// TwinCAT 3 PLC project TcTcpUdpRT_Test
// ProgramVersion: 3.1.4026.20
// libraries:
//   Tc2_Standard, * (Beckhoff Automation GmbH)
//   Tc2_System, * (Beckhoff Automation GmbH)
//   [TcTcpUdpRT], * (TcInterfaces)
//   TcUnit, * (www.tcunit.org)
// project tree:
//   / PlcTask.TcTTO, PRG_TEST.TcPOU (not stored)
//   TESTs/ ArpPing_Test.TcPOU (not stored), RingBuffer_Test.TcPOU, TcpClient_Test.TcPOU, TcpServer_Test.TcPOU, UdpSendReceive_Test.TcPOU
// real-time tasks:
//   TASK PlcTask: cycle T#1ms, priority 6, ADS port 350
// I/O:
//   DEVICE EthernetRT (RT-Ethernet Adapter)

CONFIGURATION TcTcpUdpRT_Test
    RESOURCE PLC ON TwinCAT3
        TASK PlcTask(INTERVAL := T#1ms, PRIORITY := 6);
        PROGRAM PRG_TEST WITH PlcTask : PRG_TEST;
    END_RESOURCE
END_CONFIGURATION

// ---- TESTs/RingBuffer_Test.TcPOU
FUNCTION_BLOCK RingBuffer_Test EXTENDS FB_TestSuite
VAR
	RingBuf: RingBuffer;
	RingBufUnallocated: RingBuffer;  // Init() is never called on this instance, used for the unallocated corner cases
	ReadBuffer: ARRAY[0..(TcTcpUdpRT_Param.RingBufferSize-1)] OF BYTE;
	WriteBuffer: ARRAY[0..(WriteBufferSize-1)] OF BYTE;
	emptyPointer: POINTER TO BYTE;
	bytePointer: BYTE;
END_VAR
VAR CONSTANT
	WriteBufferSize: UDINT := 35000;
END_VAR

IF NOT RingBuf.IsAllocated THEN
	RingBuf.Init(BufferSize:= TcTcpUdpRT_Param.RingBufferSize);  // Allocate once before the tests run
END_IF

//WriteWithNoDataPointer();
//WriteWithNoDataLength();
//ReadWithNoDataPointer();
//ReadWithNoDataLength();

Write3kToBufferAndEmptyIt();
ExpectBufferToBeEmpty();
ReadFromEmptyBuffer();
Write1kBytesToBuffer();
ExpectBufferNotToEmpty();

Read2kBytesFrom1kBytesBuffer();
Write25kMoreBytesToBuffer();
ExpectBufferToNotBeFull();

Read24kMoreBytesFromBuffer();
Write8kMoreBytesToBufferAndWrapAround();
Read10kMoreBytesAndWrapAround();

WriteOverflowBuffer();
WriteFullSizeOfBuffer();
ExpectBufferToBeFull();
Write1ByteOverWrapAroundAndRead1ByteOver();

// Corner cases on a buffer that was never allocated
UnallocatedBufferState();
ReadFromUnallocatedBuffer();
WriteToUnallocatedBuffer();
EmptyUnallocatedBuffer();
InitUnallocatedBufferWithDefaultSize();

METHOD EmptyUnallocatedBuffer
VAR
	Emptied: BOOL;
END_VAR
IF TEST_ORDERED('EmptyUnallocatedBuffer') THEN
	Emptied := RingBufUnallocated.EmptyBuffer();
	AssertFalse(Condition:= Emptied, Message:= 'Expected EmptyBuffer to return FALSE on an unallocated buffer');
	AssertTrue(Condition:= RingBufUnallocated.Error, Message:= 'Expected an error when emptying an unallocated buffer');
	AssertEquals_STRING(Expected:= 'Ring buffer is not allocated, call Init() first', Actual:= RingBufUnallocated.GetError, Message:= 'Unexpected error string when emptying an unallocated buffer');

	RingBufUnallocated.ResetError();
	AssertFalse(Condition:= RingBufUnallocated.Error, Message:= 'Ring buffer did not reset error after emptying unallocated buffer');
	TEST_FINISHED();
END_IF
END_METHOD

METHOD ExpectBufferNotToEmpty
IF TEST_ORDERED('ExpectBufferNotToEmpty') THEN
	AssertFalse(Condition:= RingBuf.IsBufferEmpty, Message:= 'Expected IsBufferEmpty returned TRUE when the buffer was not empty');
	TEST_FINISHED();
END_IF
END_METHOD

METHOD ExpectBufferToBeEmpty
IF TEST_ORDERED('ExpectBufferToBeEmpty') THEN
	RingBuf.EmptyBuffer();
	AssertTrue(Condition:= RingBuf.IsBufferEmpty, Message:= 'Expected IsBufferEmpty returned FALSE when the buffer was empty');
	TEST_FINISHED();
END_IF
END_METHOD

METHOD ExpectBufferToBeFull
IF TEST_ORDERED('ExpectBufferToBeFull') THEN
	AssertTRUE(Condition:= RingBuf.IsBufferFull, Message:= 'Expected IsBufferFull returned FALSE when the buffer was full');
	TEST_FINISHED();
END_IF
END_METHOD

METHOD ExpectBufferToNotBeFull
IF TEST_ORDERED('ExpectBufferToNotBeFull') THEN
	AssertFalse(Condition:= RingBuf.IsBufferFull, Message:= 'Expected IsBufferFull returned TRUE when the buffer was not full');
	TEST_FINISHED();
END_IF
END_METHOD

METHOD InitUnallocatedBufferWithDefaultSize
VAR
	DataChar: BYTE := 7;
	DataSize: UDINT := 10;
	Initialized: BOOL;
	Written: UDINT;
	Read: UDINT;
END_VAR
IF TEST_ORDERED('InitUnallocatedBufferWithDefaultSize') THEN
	// Init with size 0 falls back to the default size
	Initialized := RingBufUnallocated.Init(BufferSize:= 0);
	AssertTrue(Condition:= Initialized, Message:= 'Expected Init() with size 0 to allocate the default size');
	AssertFalse(Condition:= RingBufUnallocated.Error, Message:= RingBufUnallocated.GetError);
	AssertTrue(Condition:= RingBufUnallocated.IsAllocated, Message:= 'Expected IsAllocated to be TRUE after Init()');
	AssertEquals_UDINT(Expected:= TcTcpUdpRT_Param.RingBufferSize, Actual:= RingBufUnallocated.Size, Message:= 'Expected Size to be the default size after Init() with size 0');
	AssertTrue(Condition:= RingBufUnallocated.IsBufferEmpty, Message:= 'Expected IsBufferEmpty to be TRUE right after Init()');
	AssertFalse(Condition:= RingBufUnallocated.IsBufferFull, Message:= 'Expected IsBufferFull to be FALSE right after Init()');

	// A second Init must not reallocate or change the size
	Initialized := RingBufUnallocated.Init(BufferSize:= 123);
	AssertTrue(Condition:= Initialized, Message:= 'Expected a second Init() to return TRUE');
	AssertEquals_UDINT(Expected:= TcTcpUdpRT_Param.RingBufferSize, Actual:= RingBufUnallocated.Size, Message:= 'A second Init() changed the size of an already allocated buffer');

	// The buffer is usable after Init()
	MEMSET(destAddr:= ADR(WriteBuffer), fillByte:= DataChar, n:= DataSize);
	MEMSET(destAddr:= ADR(ReadBuffer), fillByte:= 0, n:= TcTcpUdpRT_Param.RingBufferSize);
	Written := RingBufUnallocated.Write(Data:= ADR(WriteBuffer), Length:= DataSize);
	Read := RingBufUnallocated.Read(Data:= ADR(ReadBuffer), Length:= DataSize);
	AssertEquals_UDINT(Expected:= DataSize, Actual:= Written, Message:= 'Written data to the newly allocated buffer does not match');
	AssertEquals_UDINT(Expected:= DataSize, Actual:= Read, Message:= 'Read data from the newly allocated buffer does not match');
	AssertEquals_BYTE(Expected:= DataChar, Actual:= ReadBuffer[DataSize-1], Message:= 'The last element read from the newly allocated buffer was not correct');
	AssertFalse(Condition:= RingBufUnallocated.Error, Message:= RingBufUnallocated.GetError);
	TEST_FINISHED();
END_IF
END_METHOD

METHOD Read10kMoreBytesAndWrapAround
VAR
	DataSize: UDINT := 10000;
	ExpectedSize: UDINT := 9000;
	Read: UDINT;
END_VAR
IF TEST_ORDERED('Read10kMoreBytesAndWrapAround') THEN
	MEMSET(destAddr:= ADR(ReadBuffer), fillByte:= 0, n:= TcTcpUdpRT_Param.RingBufferSize);
	
	Read := RingBuf.Read(Data:= ADR(ReadBuffer), Length:= DataSize);
	AssertEquals_UDINT(Expected:= ExpectedSize, Actual:= Read, Message:= CONCAT('Read data from ring buffer returned a length of ', TO_STRING(Read)));
	AssertTrue(Condition:= ReadBuffer[0] <> 0, Message:= 'The firste element was not different from zero');
	AssertTrue(Condition:= ReadBuffer[ExpectedSize-1] <> 0, Message:= 'The 8999th element was not different from zero');
	AssertTrue(Condition:= ReadBuffer[ExpectedSize] = 0, Message:= 'The 9000th element was not zero');
	AssertTrue(Condition:= ReadBuffer[DataSize] = 0, Message:= 'The last element was not zero');
	TEST_FINISHED();
END_IF
END_METHOD

METHOD Read24kMoreBytesFromBuffer
VAR
	DataSize: UDINT := 24000;
	ExpectedSize: UDINT := 24000;
	Read: UDINT;
END_VAR
IF TEST_ORDERED('Read24kMoreBytesFromBuffer') THEN
	MEMSET(destAddr:= ADR(ReadBuffer), fillByte:= 0, n:= TcTcpUdpRT_Param.RingBufferSize);
	
	Read := RingBuf.Read(Data:= ADR(ReadBuffer), Length:= DataSize);
	AssertEquals_UDINT(Expected:= ExpectedSize, Actual:= Read, Message:= CONCAT('Read data from ring buffer returned a length of ', TO_STRING(Read)));
	AssertTrue(Condition:= ReadBuffer[0] <> 0, Message:= 'The firste element was not different from zero');
	AssertTrue(Condition:= ReadBuffer[18475] <> 0, Message:= 'A random element was not different from zero');
	AssertTrue(Condition:= ReadBuffer[DataSize-1] <> 0, Message:= 'The last element was not different from zero');
	TEST_FINISHED();
END_IF
END_METHOD

METHOD Read2kBytesFrom1kBytesBuffer
VAR
	DataSize: UDINT := 2000;
	ExpectedSize: UDINT := 1000;
	Read: UDINT;
END_VAR
IF TEST_ORDERED('Read2kBytesFrom1kBytesBuffer') THEN
	MEMSET(destAddr:= ADR(ReadBuffer), fillByte:= 0, n:= TcTcpUdpRT_Param.RingBufferSize);
	
	Read := RingBuf.Read(Data:= ADR(ReadBuffer), Length:= DataSize);
	AssertEquals_UDINT(Expected:= ExpectedSize, Actual:= Read, Message:= CONCAT('Read data from ring buffer returned a length of ', TO_STRING(Read)));
	AssertTrue(Condition:= ReadBuffer[0] <> 0, Message:= 'The firste element was not different from zero');
	AssertTrue(Condition:= ReadBuffer[ExpectedSize-1] <> 0, Message:= 'The 999th element was not different from zero');
	AssertTrue(Condition:= ReadBuffer[ExpectedSize] = 0, Message:= 'The 1000th element was not zero');
	AssertTrue(Condition:= ReadBuffer[DataSize-1] = 0, Message:= 'The last element was not zero');
	TEST_FINISHED();
END_IF
END_METHOD

METHOD ReadFromEmptyBuffer
VAR
	DataSize: UDINT := 10;
	ExpectedSize: UDINT := 0;
	Read: UDINT;
END_VAR
IF TEST_ORDERED('ReadFromEmptyBuffer') THEN
	MEMSET(destAddr:= ADR(ReadBuffer), fillByte:= 0, n:= TcTcpUdpRT_Param.RingBufferSize);
	
	Read := RingBuf.Read(Data:= ADR(ReadBuffer), Length:= DataSize);
	AssertEquals_UDINT(Expected:= ExpectedSize, Actual:= Read, Message:= CONCAT('Read data from empty ring buffer returned a length of ', TO_STRING(Read)));
	TEST_FINISHED();
END_IF
END_METHOD

METHOD ReadFromUnallocatedBuffer
VAR
	DataSize: UDINT := 10;
	Read: UDINT;
END_VAR
IF TEST_ORDERED('ReadFromUnallocatedBuffer') THEN
	MEMSET(destAddr:= ADR(ReadBuffer), fillByte:= 0, n:= TcTcpUdpRT_Param.RingBufferSize);

	Read := RingBufUnallocated.Read(Data:= ADR(ReadBuffer), Length:= DataSize);
	AssertEquals_UDINT(Expected:= 0, Actual:= Read, Message:= CONCAT('Read from unallocated ring buffer returned a length of ', TO_STRING(Read)));
	AssertTrue(Condition:= RingBufUnallocated.Error, Message:= 'Expected an error when reading from an unallocated buffer');
	AssertEquals_STRING(Expected:= 'Ring buffer is not allocated, call Init() first', Actual:= RingBufUnallocated.GetError, Message:= 'Unexpected error string when reading from an unallocated buffer');
	AssertEquals_BYTE(Expected:= 0, Actual:= ReadBuffer[0], Message:= 'Read from unallocated buffer modified the destination');

	RingBufUnallocated.ResetError();
	AssertFalse(Condition:= RingBufUnallocated.Error, Message:= 'Ring buffer did not reset error after read from unallocated buffer');
	TEST_FINISHED();
END_IF
END_METHOD

METHOD ReadWithNoDataLength
IF TEST_ORDERED('ReadWithNoDataLength') THEN
	emptyPointer := ADR(bytePointer);
	RingBuf.Read(Data:= emptyPointer, Length:= 0);
	AssertTrue(Condition:= RingBuf.Error, Message:= 'Reading to ring buffer did not handle a data length of zero');
	RingBuf.ResetError();
	TEST_FINISHED();
END_IF
END_METHOD

METHOD ReadWithNoDataPointer
IF TEST_ORDERED('ReadWithNoDataPointer') THEN
	emptyPointer := 0;
	RingBuf.Read(Data:= emptyPointer, Length:= 10);
	AssertTrue(Condition:= RingBuf.Error, Message:= 'Reading to ring buffer did not handle empty data pointer');
	RingBuf.ResetError();
	TEST_FINISHED();
END_IF
END_METHOD

METHOD UnallocatedBufferState
IF TEST_ORDERED('UnallocatedBufferState') THEN
	AssertFalse(Condition:= RingBufUnallocated.IsAllocated, Message:= 'Expected IsAllocated to be FALSE before Init()');
	AssertEquals_UDINT(Expected:= 0, Actual:= RingBufUnallocated.Size, Message:= 'Expected Size to be 0 before Init()');
	AssertTrue(Condition:= RingBufUnallocated.IsBufferEmpty, Message:= 'Expected IsBufferEmpty to be TRUE for an unallocated buffer');
	AssertFalse(Condition:= RingBufUnallocated.IsBufferFull, Message:= 'Expected IsBufferFull to be FALSE for an unallocated buffer');
	AssertFalse(Condition:= RingBufUnallocated.Error, Message:= 'Expected no error on an unallocated buffer that has not been used');
	TEST_FINISHED();
END_IF
END_METHOD

METHOD Write1ByteOverWrapAroundAndRead1ByteOver
VAR
	DataChar1: BYTE := 55;
	DataSize1: UDINT := TcTcpUdpRT_Param.RingBufferSize - 10;
	ExpectedSize1: UDINT := TcTcpUdpRT_Param.RingBufferSize - 10;
	
	DataChar2: BYTE := 57;
	DataSize2: UDINT := 11;
	ExpectedSize2: UDINT := 11;
	
	Written: UDINT;
	Read: UDINT;
END_VAR
IF TEST_ORDERED('Write1ByteOverWrapAroundAndRead1ByteOver') THEN
	RingBuf.EmptyBuffer();
	MEMSET(destAddr:= ADR(WriteBuffer), fillByte:= DataChar1, n:= DataSize1);
	MEMSET(destAddr:= ADR(ReadBuffer), fillByte:= 0, n:= TcTcpUdpRT_Param.RingBufferSize);
	Written := RingBuf.Write(Data:= ADR(WriteBuffer), Length:= DataSize1);
	Read := RingBuf.Read(Data:= ADR(ReadBuffer), Length:= DataSize1);
	AssertEquals_UDINT(Expected:= ExpectedSize1, Actual:= Written, Message:= 'Written data to ring buffer does not match actual');
	AssertEquals_UDINT(Expected:= ExpectedSize1, Actual:= Read, Message:= CONCAT('Read data from ring buffer returned a length of ', TO_STRING(Read)));
	
	
	MEMSET(destAddr:= ADR(WriteBuffer), fillByte:= DataChar2, n:= DataSize2);
	MEMSET(destAddr:= ADR(ReadBuffer), fillByte:= 0, n:= TcTcpUdpRT_Param.RingBufferSize);
	Written := RingBuf.Write(Data:= ADR(WriteBuffer), Length:= DataSize2);
	Read := RingBuf.Read(Data:= ADR(ReadBuffer), Length:= DataSize2);
	AssertEquals_UDINT(Expected:= ExpectedSize2, Actual:= Written, Message:= 'Written data to ring buffer does not match actual');
	AssertEquals_UDINT(Expected:= ExpectedSize2, Actual:= Read, Message:= CONCAT('Read data from ring buffer returned a length of ', TO_STRING(Read)));
	AssertEquals_BYTE(Expected:= DataChar2, Actual:= ReadBuffer[ExpectedSize2-2], Message:= 'The element before wrap around was not correct');
	AssertEquals_BYTE(Expected:= DataChar2, Actual:= ReadBuffer[ExpectedSize2-1], Message:= 'The element after wrap around was not correct');
	AssertEquals_BYTE(Expected:= 0, Actual:= ReadBuffer[ExpectedSize2], Message:= 'The element after last was not zero');
	TEST_FINISHED();
END_IF
END_METHOD

METHOD Write1kBytesToBuffer
VAR
	DataChar: BYTE := 3;
	DataSize: UDINT := 1000;
	ExpectedSize: UDINT := 1000;
	Written: UDINT;
END_VAR
IF TEST_ORDERED('Write1kBytesToBuffer') THEN
	MEMSET(destAddr:= ADR(WriteBuffer), fillByte:= DataChar, n:= DataSize);
	
	Written := RingBuf.Write(Data:= ADR(WriteBuffer), Length:= DataSize);
	AssertEquals_UDINT(Expected:= ExpectedSize, Actual:= Written, Message:= 'Written data to ring buffer does not match actual');
	TEST_FINISHED();
END_IF
END_METHOD

METHOD Write25kMoreBytesToBuffer
VAR
	DataChar: BYTE := 8;
	DataSize: UDINT := 25000;
	ExpectedSize: UDINT := 25000;
	Written: UDINT;
END_VAR
IF TEST_ORDERED('Write25kMoreBytesToBuffer') THEN
	MEMSET(destAddr:= ADR(WriteBuffer), fillByte:= DataChar, n:= DataSize);
	
	Written := RingBuf.Write(Data:= ADR(WriteBuffer), Length:= DataSize);
	AssertEquals_UDINT(Expected:= ExpectedSize, Actual:= Written, Message:= 'Written data to ring buffer does not match actual');
	TEST_FINISHED();
END_IF
END_METHOD

METHOD Write3kToBufferAndEmptyIt
VAR
	DataChar: BYTE := 69;
	DataSize: UDINT := 3000;
	ExpectedSize: UDINT := 3000;
	Written: UDINT;
END_VAR
IF TEST_ORDERED('Write3kToBufferAndEmptyIt') THEN
	MEMSET(destAddr:= ADR(WriteBuffer), fillByte:= DataChar, n:= DataSize);
	
	AssertTrue(Condition:= RingBuf.IsBufferEmpty, Message:= 'Expected IsBufferEmpty returned FALSE when the buffer was empty');
	Written := RingBuf.Write(Data:= ADR(WriteBuffer), Length:= DataSize);
	AssertEquals_UDINT(Expected:= ExpectedSize, Actual:= Written, Message:= 'Written data to ring buffer does not match actual');
	AssertFalse(Condition:= RingBuf.IsBufferEmpty, Message:= 'Expected IsBufferEmpty returned TRUE when the buffer was not empty');
	
	RingBuf.EmptyBuffer();
	AssertTrue(Condition:= RingBuf.IsBufferEmpty, Message:= 'Expected IsBufferEmpty returned FALSE when the buffer was empty');
	TEST_FINISHED();
END_IF
END_METHOD

METHOD Write8kMoreBytesToBufferAndWrapAround
VAR
	DataChar: BYTE := 16;
	DataSize: UDINT := 8000;
	ExpectedSize: UDINT := 8000;
	Written: UDINT;
END_VAR
IF TEST_ORDERED('Write8kMoreBytesToBufferAndWrapAround') THEN
	MEMSET(destAddr:= ADR(WriteBuffer), fillByte:= DataChar, n:= DataSize);
	
	Written := RingBuf.Write(Data:= ADR(WriteBuffer), Length:= DataSize);
	AssertEquals_UDINT(Expected:= ExpectedSize, Actual:= Written, Message:= 'Written data to ring buffer does not match actual');
	TEST_FINISHED();
END_IF
END_METHOD

METHOD WriteFullSizeOfBuffer
VAR
	DataChar: BYTE := 24;
	DataSize: UDINT := TcTcpUdpRT_Param.RingBufferSize-1;
	ExpectedSize: UDINT := TcTcpUdpRT_Param.RingBufferSize-1;
	Written: UDINT;
END_VAR
IF TEST_ORDERED('WriteFullSizeOfBuffer') THEN
	MEMSET(destAddr:= ADR(WriteBuffer), fillByte:= DataChar, n:= DataSize);
	
	Written := RingBuf.Write(Data:= ADR(WriteBuffer), Length:= DataSize);
	AssertEquals_UDINT(Expected:= ExpectedSize, Actual:= Written, Message:= 'Written data to ring buffer does not match actual');
	AssertTrue(Condition:= RingBuf.IsBufferFull, Message:= 'Ring buffer was not full after writing full size');
	TEST_FINISHED();
END_IF
END_METHOD

METHOD WriteOverflowBuffer
VAR
	DataChar: BYTE := 16;
	DataSize: UDINT := WriteBufferSize;
	Written: UDINT;
END_VAR
IF TEST_ORDERED('WriteOverflowBuffer') THEN
	MEMSET(destAddr:= ADR(WriteBuffer), fillByte:= DataChar, n:= DataSize);
	
	Written := RingBuf.Write(Data:= ADR(WriteBuffer), Length:= DataSize);
	AssertTrue(Condition:= RingBuf.Error, Message:= RingBuf.GetError);
	RingBuf.ResetError();
	AssertFalse(Condition:= RingBuf.Error, Message:= 'Ring buffer did not reset error after overflow');
	TEST_FINISHED();
END_IF
END_METHOD

METHOD WriteToUnallocatedBuffer
VAR
	DataChar: BYTE := 42;
	DataSize: UDINT := 10;
	Written: UDINT;
END_VAR
IF TEST_ORDERED('WriteToUnallocatedBuffer') THEN
	MEMSET(destAddr:= ADR(WriteBuffer), fillByte:= DataChar, n:= DataSize);

	Written := RingBufUnallocated.Write(Data:= ADR(WriteBuffer), Length:= DataSize);
	AssertEquals_UDINT(Expected:= 0, Actual:= Written, Message:= CONCAT('Write to unallocated ring buffer returned a length of ', TO_STRING(Written)));
	AssertTrue(Condition:= RingBufUnallocated.Error, Message:= 'Expected an error when writing to an unallocated buffer');
	AssertEquals_STRING(Expected:= 'Ring buffer is not allocated, call Init() first', Actual:= RingBufUnallocated.GetError, Message:= 'Unexpected error string when writing to an unallocated buffer');
	AssertTrue(Condition:= RingBufUnallocated.IsBufferEmpty, Message:= 'Expected IsBufferEmpty to stay TRUE after a rejected write');

	RingBufUnallocated.ResetError();
	AssertFalse(Condition:= RingBufUnallocated.Error, Message:= 'Ring buffer did not reset error after write to unallocated buffer');
	TEST_FINISHED();
END_IF
END_METHOD

METHOD WriteWithNoDataLength
IF TEST_ORDERED('WriteWithNoDataLength') THEN
	emptyPointer := ADR(bytePointer);
	RingBuf.Write(Data:= emptyPointer, Length:= 0);
	AssertTrue(Condition:= RingBuf.Error, Message:= 'Writing to ring buffer did not handle a data length of zero');
	RingBuf.ResetError();
	TEST_FINISHED();
END_IF
END_METHOD

METHOD WriteWithNoDataPointer
IF TEST_ORDERED('WriteWithNoDataPointer') THEN
	emptyPointer := 0;
	RingBuf.Write(Data:= emptyPointer, Length:= 10);
	AssertTrue(Condition:= RingBuf.Error, Message:= 'Writing to ring buffer did not handle empty data pointer');
	RingBuf.ResetError();
	TEST_FINISHED();
END_IF
END_METHOD

END_FUNCTION_BLOCK

// ---- TESTs/TcpClient_Test.TcPOU
FUNCTION_BLOCK TcpClient_Test EXTENDS FB_TestSuite
VAR
	startTcpClientTest		: BOOL;
	tcpClientTestDone		: BOOL;
	tcpServerTestTimeout	: TON := (PT:= T#2M);
	
	tcpClient	: TcTcpClient(BufferSize:= TcTcpUdpRT_Param.RingBufferSize);
	serverAddr	: STRING(15) := '192.168.1.119';
	serverPort	: UINT := 9901;
	txData		: STRING(25) := 'Hello from PLC TCP client';
	txCounter	: UDINT;
	rxData		: STRING;
	rxCounter	: UDINT;
	methodTimeout	: TON;
END_VAR

tcpClient.Run();

IF startTcpClientTest THEN
	ConnectToTcpServer();
	SendMessageToTcpServer();
	ReceiveMessageFromTcpServer();
	CloseConnectionToTcpServer();
END_IF

TEST('RunTcpClientTest');
tcpServerTestTimeout(IN:= startTcpClientTest);
IF tcpClientTestDone THEN
	tcpServerTestTimeout(IN:= FALSE);
	TEST_FINISHED();
ELSIF tcpServerTestTimeout.Q THEN
	AssertFalse(Condition:= tcpServerTestTimeout.Q, Message:= 'TcpClient_Test timed out while running');
	tcpServerTestTimeout(IN:= FALSE);
	TEST_FINISHED();
ELSIF tcpClient.Error THEN
	AssertFalse(Condition:= tcpClient.Error, Message:= tcpClient.GetError);
	tcpServerTestTimeout(IN:= FALSE);
	TEST_FINISHED();
END_IF

METHOD CloseConnectionToTcpServer
VAR_INST
	delay: TIME := T#15S;
END_VAR
IF TEST_ORDERED('CloseConnectionToTcpServer') THEN
	methodTimeout(IN:= TRUE, PT:= delay);
	IF tcpClient.Disconnect() THEN
		tcpClientTestDone := TRUE;
		methodTimeout(IN:= FALSE);
		TEST_FINISHED();
	ELSIF methodTimeout.Q THEN
		AssertTrue(Condition:= FALSE, Message:= 'TCP client timed out disconnecting from the TCP server');
		methodTimeout(IN:= FALSE);
		TEST_FINISHED();
	END_IF
END_IF
END_METHOD

METHOD ConnectToTcpServer
VAR_INST
	delay: TIME := T#15S;
END_VAR
IF TEST_ORDERED('ConnectToTcpServer') THEN
	methodTimeout(IN:= TRUE, PT:= delay);
	IF tcpClient.Connect(IpAddress:= serverAddr, Port:= serverPort) THEN
		methodTimeout(IN:= FALSE);
		TEST_FINISHED();
	ELSIF methodTimeout.Q THEN
		AssertTrue(Condition:= FALSE, Message:= 'TCP client timed out connecting to the TCP server');
		methodTimeout(IN:= FALSE);
		TEST_FINISHED();
	END_IF
END_IF
END_METHOD

METHOD ReceiveMessageFromTcpServer
VAR_INST
	delay: TIME := T#15S;
END_VAR
IF TEST_ORDERED('ReceiveMessageFromTcpServer') THEN
	methodTimeout(IN:= TRUE, PT:= delay);
	IF tcpClient.IsDataAvailable THEN
		IF tcpClient.Receive(DataPointer:= ADR(rxData), DataLength:= SIZEOF(rxData), ReceivedLength=> rxCounter) THEN
			ADSLOGSTR(msgCtrlMask:= ADSLOG_MSGTYPE_LOG, msgFmtStr:= 'Message received: %s', strArg:= rxData);
			AssertTrue(Condition:= rxCounter > 0, Message:= 'The data from the TCP server had a length of zero');
			methodTimeout(IN:= FALSE);
			TEST_FINISHED();
		END_IF
	ELSIF methodTimeout.Q THEN
		AssertTrue(Condition:= FALSE, Message:= 'TCP client timed out waiting for data from the TCP server');
		methodTimeout(IN:= FALSE);
		TEST_FINISHED();
	END_IF
END_IF
END_METHOD

METHOD SendMessageToTcpServer
VAR_INST
	delay: TIME := T#15S;
END_VAR
IF TEST_ORDERED('SendMessageToTcpServer') THEN
	methodTimeout(IN:= TRUE, PT:= delay);
	IF tcpClient.Send(DataPointer:= ADR(txData), DataLength:= SIZEOF(txData), DataSent=> txCounter) THEN
		ADSLOGSTR(msgCtrlMask:= ADSLOG_MSGTYPE_LOG, msgFmtStr:= 'Message sent: %s', strArg:= txData);
		AssertTrue(Condition:= txCounter > 0, Message:= 'The data sent to the TCP server had a length of zero');
		methodTimeout(IN:= FALSE);
		TEST_FINISHED();
	ELSIF methodTimeout.Q THEN
		AssertTrue(Condition:= FALSE, Message:= 'TCP client timed out sending data to the TCP server');
		methodTimeout(IN:= FALSE);
		TEST_FINISHED();
	END_IF
END_IF
END_METHOD

END_FUNCTION_BLOCK

// ---- TESTs/TcpServer_Test.TcPOU
FUNCTION_BLOCK TcpServer_Test EXTENDS FB_TestSuite
VAR
	startTcpServerTest		: BOOL;
	tcpServerTestDone		: BOOL;
	tcpServerTestTimeout	: TON := (PT:= T#2M);
	
	tcpServer	: TcTcpServer(BufferSize:= TcTcpUdpRT_Param.RingBufferSize);
	listenPort	: UINT := 9900;
	txData		: STRING(25) := 'Hello from PLC TCP server';
	txCounter	: UDINT;
	rxData		: STRING;
	rxCounter	: UDINT;
	methodTimeout		: TON;
END_VAR

tcpServer.Run();

IF startTcpServerTest THEN
	OpenConnectionAndListenForClient();
	WaitForTcpClientToConnect();
	ReceiveDataFromTcpClient();
	SendDataToTcpClient();
	WaitForClientToDisconnect();
END_IF

TEST('RunTcpServerTest');
tcpServerTestTimeout(IN:= startTcpServerTest);
IF tcpServerTestDone THEN
	tcpServerTestTimeout(IN:= FALSE);
	TEST_FINISHED();
ELSIF tcpServerTestTimeout.Q THEN
	AssertFalse(Condition:= tcpServerTestTimeout.Q, Message:= 'TcpServer_Test timed out while running');
	tcpServerTestTimeout(IN:= FALSE);
	TEST_FINISHED();
ELSIF tcpServer.Error THEN
	AssertFalse(Condition:= tcpServer.Error, Message:= tcpServer.GetError);
	tcpServerTestTimeout(IN:= FALSE);
	TEST_FINISHED();
END_IF

METHOD OpenConnectionAndListenForClient
VAR_INST
	openConnection: BOOL;
END_VAR
IF TEST_ORDERED('OpenConnectionAndListenForClient') THEN
	openConnection := tcpServer.OpenConnection(listenPort);
	AssertTrue(Condition:= openConnection, Message:= 'Failed to open TCP server connection');
	TEST_FINISHED();	
END_IF
END_METHOD

METHOD ReceiveDataFromTcpClient
VAR_INST
	delay: TIME := T#15S;
END_VAR
IF TEST_ORDERED('ReceiveDataFromTcpClient') THEN
	methodTimeout(IN:= TRUE, PT:= delay);
	IF tcpServer.IsDataAvailable THEN
		IF tcpServer.Receive(DataPointer:= ADR(rxData), DataLength:= SIZEOF(rxData), ReceivedLength=> rxCounter) THEN
			ADSLOGSTR(msgCtrlMask:= ADSLOG_MSGTYPE_LOG, msgFmtStr:= 'Message received: %s', strArg:= rxData);
			AssertTrue(Condition:= rxCounter > 0, Message:= 'The data from the TCP client had a length of zero');
			methodTimeout(IN:= FALSE);
			TEST_FINISHED();
		END_IF
	ELSIF methodTimeout.Q THEN
		AssertTrue(Condition:= FALSE, Message:= 'TCP server timed out waiting for data from the TCP client');
		methodTimeout(IN:= FALSE);
		TEST_FINISHED();
	END_IF
END_IF
END_METHOD

METHOD SendDataToTcpClient
VAR_INST
	delay: TIME := T#15S;
END_VAR
IF TEST_ORDERED('SendDataToTcpClient') THEN
	methodTimeout(IN:= TRUE, PT:= delay);
	IF tcpServer.Send(DataPointer:= ADR(txData), DataLength:= SIZEOF(txData), DataSent=> txCounter) THEN
		ADSLOGSTR(msgCtrlMask:= ADSLOG_MSGTYPE_LOG, msgFmtStr:= 'Message sent: %s', strArg:= txData);
		AssertTrue(Condition:= txCounter > 0, Message:= 'The data sent to the TCP client had a length of zero');
		methodTimeout(IN:= FALSE);
		TEST_FINISHED();
	ELSIF methodTimeout.Q THEN
		AssertTrue(Condition:= FALSE, Message:= 'TCP server timed out sending data to the TCP client');
		methodTimeout(IN:= FALSE);
		TEST_FINISHED();
	END_IF
END_IF
END_METHOD

METHOD WaitForClientToDisconnect
VAR_INST
	delay: TIME := T#15S;
END_VAR
IF TEST_ORDERED('WaitForClientToDisconnect') THEN
	methodTimeout(IN:= TRUE, PT:= delay);
	IF NOT  tcpServer.IsConnected THEN
		tcpServerTestDone := TRUE;
		methodTimeout(IN:= FALSE);
		TEST_FINISHED();
	ELSIF methodTimeout.Q THEN
		AssertTrue(Condition:= FALSE, Message:= 'TCP server timed out waiting for TCP client to disconnection');
		methodTimeout(IN:= FALSE);
		TEST_FINISHED();
	END_IF
END_IF
END_METHOD

METHOD WaitForTcpClientToConnect
VAR_INST
	delay: TIME := T#15S;
END_VAR
IF TEST_ORDERED('WaitForTcpClientToConnect') THEN
	methodTimeout(IN:= TRUE, PT:= delay);
	IF tcpServer.IsConnected THEN
		methodTimeout(IN:= FALSE);
		TEST_FINISHED();
	ELSIF methodTimeout.Q THEN
		AssertTrue(Condition:= FALSE, Message:= 'TCP server timed out waiting for the TCP client to connection');
		methodTimeout(IN:= FALSE);
		TEST_FINISHED();
	END_IF
END_IF
END_METHOD

END_FUNCTION_BLOCK

// ---- TESTs/UdpSendReceive_Test.TcPOU
FUNCTION_BLOCK UdpSendReceive_Test EXTENDS FB_TestSuite
VAR
	startUdpTest		: BOOL;
	udpTestDone			: BOOL;
	waitListenTestDone	: BOOL;
	tcpServerTestTimeout	: TON := (PT:= T#2M);
	
	udpClient		: TcUdpSendReceive(BufferSize:= TcTcpUdpRT_Param.RingBufferSize);
	clientAddr		: STRING(15) := '192.168.1.119';
	listenPort		: UINT := 9902;
	sendPort		: UINT := 9901;
	txData			: STRING(25) := 'Hello from PLC UDP client';
	txCounter		: UDINT;
	rxData			: STRING;
	rxCounter		: UDINT;
	methodTimeout	: TON;
END_VAR

udpClient.Run();

IF startUdpTest THEN
	ListenOnUdpPort();
	ReceiveUdpMessage();
	SendUdpMessage();
END_IF

TEST('RunUdpClientTest');
tcpServerTestTimeout(IN:= startUdpTest);
IF udpTestDone THEN
	tcpServerTestTimeout(IN:= FALSE);
	TEST_FINISHED();
ELSIF tcpServerTestTimeout.Q THEN
	AssertFalse(Condition:= tcpServerTestTimeout.Q, Message:= 'UdpClient_Test timed out while running');
	tcpServerTestTimeout(IN:= FALSE);
	TEST_FINISHED();
ELSIF udpClient.Error THEN
	AssertFalse(Condition:= udpClient.Error, Message:= udpClient.GetError);
	tcpServerTestTimeout(IN:= FALSE);
	TEST_FINISHED();
END_IF

METHOD ListenOnUdpPort
VAR_INST
	delay: TIME := T#15S;
END_VAR
IF TEST_ORDERED('ListenOnUdpPort') THEN
	methodTimeout(IN:= TRUE, PT:= delay);
	IF udpClient.StartListen(Port:= listenPort) THEN
		ADSLOGDINT(msgCtrlMask:= ADSLOG_MSGTYPE_LOG, msgFmtStr:= 'UDP client listening on port %d', dintArg:= listenPort);
		waitListenTestDone := TRUE;
		methodTimeout(IN:= FALSE);
		TEST_FINISHED();
	ELSIF methodTimeout.Q THEN
		AssertTrue(Condition:= FALSE, Message:= 'UDP client timed out listening on port');
		methodTimeout(IN:= FALSE);
		TEST_FINISHED();
	END_IF
END_IF
END_METHOD

METHOD ReceiveUdpMessage
VAR_INST
	delay: TIME := T#15S;
END_VAR
IF TEST_ORDERED('ReceiveUdpMessage') THEN
	methodTimeout(IN:= TRUE, PT:= delay);
	IF udpClient.IsDataAvailable THEN
		IF udpClient.Receive(DataPointer:= ADR(rxData), DataLength:= SIZEOF(rxData), ReceivedLength=> rxCounter) THEN
			ADSLOGSTR(msgCtrlMask:= ADSLOG_MSGTYPE_LOG, msgFmtStr:= 'UDP message received: %s', strArg:= rxData);
			AssertTrue(Condition:= rxCounter > 0, Message:= 'The data from the UDP server had a length of zero');
			methodTimeout(IN:= FALSE);
			TEST_FINISHED();
		END_IF
	ELSIF methodTimeout.Q THEN
		AssertTrue(Condition:= FALSE, Message:= 'UDP client timed out waiting for data from the UDP server');
		methodTimeout(IN:= FALSE);
		TEST_FINISHED();
	END_IF
END_IF
END_METHOD

METHOD SendUdpMessage
VAR_INST
	delay: TIME := T#15S;
	i: INT;
END_VAR
IF TEST_ORDERED('SendUdpMessage') THEN
	methodTimeout(IN:= TRUE, PT:= delay);
	IF udpClient.Send(IpAddress:= clientAddr, Port:= sendPort, DataPointer:= ADR(txData), DataLength:= SIZEOF(txData)) THEN
		ADSLOGSTR(msgCtrlMask:= ADSLOG_MSGTYPE_LOG, msgFmtStr:= 'UDP message sent: %s', strArg:= txData);
		udpTestDone := TRUE;
		methodTimeout(IN:= FALSE);
		TEST_FINISHED();
	ELSIF methodTimeout.Q THEN
		AssertTrue(Condition:= FALSE, Message:= 'UDP client timed out sending data to the UDP server');
		methodTimeout(IN:= FALSE);
		TEST_FINISHED();
	END_IF
END_IF
END_METHOD

END_FUNCTION_BLOCK
